// TIA Portal V16 export
// export: Created 2022-09-01T14:29:23.8061555Z, ExportSetting WithDefaults, DisplayName Totally Integrated Automation Portal, DisplayVersion V16, DisplayName TIA Portal Version Control Interface, DisplayVersion V16, DisplayName TIA Portal Openness, DisplayVersion V16, DisplayName STEP 7 Professional, DisplayVersion V16, DisplayName STEP 7 Safety, DisplayVersion V16, DisplayName WinCC Advanced, DisplayVersion V16
DATA_BLOCK "Info_Ciclo"   // DB10
{ S7_Optimized_Access := 'TRUE' }
VERSION : 0.1
// stored: AutoNumber true, IsOnlyStoredInLoadMemory false, IsRetainMemResEnabled false, IsWriteProtectedInAS false, MemoryReserve 100
   VAR RETAIN
      LS101_SR : Bool;
   END_VAR
   VAR
      ESTADO_CICLO : Bool;
      CONTAGEM_CICLOS : Int;
      LIMITE_CONTAGEM : Bool;
   END_VAR
BEGIN
END_DATA_BLOCK
